FUNCTION F_Scale : INT
VAR_INPUT
END_VAR
VAR
END_VAR

END_FUNCTION

(* stored: Version 1.1.0.1, ProductVersion 3.1.4020.14
   POU F_Scale: Id {76bd311d-7d8e-4dcc-8617-1a719685d0d2}, SpecialFunc None *)
